// TIA Portal V17 export
// export: Created 2025-04-11T04:54:23.7886703Z, ExportSetting WithDefaults, DisplayName Totally Integrated Automation Portal, DisplayVersion V17, DisplayName TIA Portal Openness, DisplayVersion V17, DisplayName TIA Portal Version Control Interface, DisplayVersion V17, DisplayName SINAMICS Startdrive Advanced, DisplayVersion V17, DisplayName SINAMICS Startdrive G130, G150, S120, S150, SINAMICS MV, S210, DisplayVersion V17, DisplayName SINAMICS Startdrive G110M, G120, G120C, G120D, G120P, G115D, DisplayVersion V17, DisplayName STEP 7 Professional, DisplayVersion V17, DisplayName STEP 7 Safety, DisplayVersion V17, DisplayName WinCC Advanced, DisplayVersion V17
TYPE "UDT_Valve_ALM"
// stored: IsFailsafeCompliant false
   STRUCT
      OUT_wALM : Word;   // 报警字 (Bit0=开阀超时报警, Bit1=关阀超时报警, Bit2=传感器故障报警)
      OUT_xSensorFault : Bool;   // 传感器故障
      OUT_xOpenTimeout : Bool;   // 开阀超时
      OUT_xCloseTimeout : Bool;   // 关阀超时
   END_STRUCT;
END_TYPE
